FUNCTION_BLOCK WaterTankSystem
  (* Standard: 61499-2 *)
  (* Version 0.1, 2015-00-11, syy, syy-PC *)
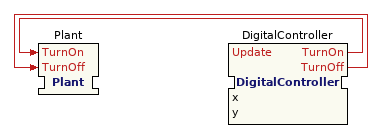
  FBS
    DigitalController : DigitalController;
    Plant : Plant;
  END_FBS
  EVENT_CONNECTIONS
    DigitalController.TurnOn TO Plant.TurnOn;
    DigitalController.TurnOff TO Plant.TurnOff;
  END_CONNECTIONS
END_FUNCTION_BLOCK
